FUNCTION_BLOCK FB_FT_PIDWL (* Composite Function Block Type *)
  (* Standard: 61499-2 *)
  (* Version 0.0, 2013-10-19, 4DIAC-IDE, 4DIAC-Consortium *)
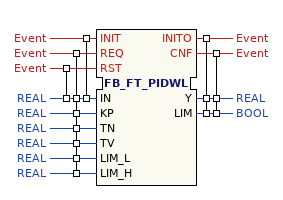
  EVENT_INPUT
    INIT WITH IN; (* Initialization Request *)
    REQ WITH IN, LIM_H, LIM_L, TV, TN, KP; (* Normal Execution Request *)
    RST WITH IN;
  END_EVENT
  EVENT_OUTPUT
    INITO WITH Y, LIM; (* Initialization Confirm *)
    CNF WITH Y, LIM; (* Execution Confirmation *)
  END_EVENT
  VAR_INPUT
    IN : REAL; (* Input event qualifier *)
    KP : REAL := 1.0;
    TN : REAL := 1.0;
    TV : REAL := 1.0;
    LIM_L : REAL := -1.0E38;
    LIM_H : REAL := 1.0E38;
  END_VAR
  VAR_OUTPUT
    Y : REAL; (* Output event qualifier *)
    LIM : BOOL;
  END_VAR
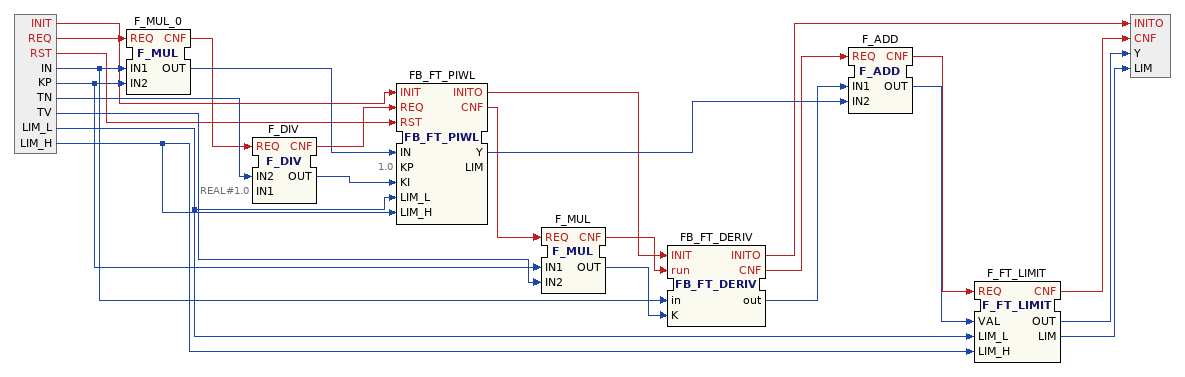
  FBS
    FB_FT_PIWL : FB_FT_PIWL(KP := 1.0);
    FB_FT_DERIV : FB_FT_DERIV;
    F_ADD : F_ADD;
    F_MUL : F_MUL;
    F_MUL_0 : F_MUL;
    F_DIV : F_DIV(IN1 := REAL#1.0);
    F_FT_LIMIT : F_FT_LIMIT;
  END_FBS
  EVENT_CONNECTIONS
    INIT TO FB_FT_PIWL.INIT;
    FB_FT_PIWL.INITO TO FB_FT_DERIV.INIT;
    FB_FT_DERIV.INITO TO INITO;
    F_MUL.CNF TO FB_FT_DERIV.run;
    FB_FT_PIWL.CNF TO F_MUL.REQ;
    RST TO FB_FT_PIWL.RST;
    REQ TO F_MUL_0.REQ;
    F_MUL_0.CNF TO F_DIV.REQ;
    F_DIV.CNF TO FB_FT_PIWL.REQ;
    FB_FT_DERIV.CNF TO F_ADD.REQ;
    F_ADD.CNF TO F_FT_LIMIT.REQ;
    F_FT_LIMIT.CNF TO CNF;
  END_CONNECTIONS
  DATA_CONNECTIONS
    LIM_L TO FB_FT_PIWL.LIM_L;
    LIM_H TO FB_FT_PIWL.LIM_H;
    FB_FT_DERIV.out TO F_ADD.IN1;
    FB_FT_PIWL.Y TO F_ADD.IN2;
    F_MUL.OUT TO FB_FT_DERIV.K;
    IN TO FB_FT_DERIV.in;
    KP TO F_MUL.IN1;
    TV TO F_MUL.IN2;
    F_MUL_0.OUT TO FB_FT_PIWL.IN;
    IN TO F_MUL_0.IN1;
    KP TO F_MUL_0.IN2;
    F_DIV.OUT TO FB_FT_PIWL.KI;
    TN TO F_DIV.IN2;
    F_FT_LIMIT.OUT TO Y;
    F_ADD.OUT TO F_FT_LIMIT.VAL;
    F_FT_LIMIT.LIM TO LIM;
    LIM_L TO F_FT_LIMIT.LIM_L;
    LIM_H TO F_FT_LIMIT.LIM_H;
  END_CONNECTIONS
END_FUNCTION_BLOCK
